FUNCTION_BLOCK FB_Toggle

VAR
	fbTon : TON := (PT := T#10S);
	bStart : BOOL := TRUE;
	fbTof : TOF := (PT := T#10S);
END_VAR

fbTon(IN := bStart);
IF fbTon.Q THEN
	bStart := FALSE;
END_IF
fbTof (IN := bStart);	
IF NOT fbTof.Q	THEN
	bStart := TRUE;
END_IF

END_FUNCTION_BLOCK

(* stored: Version 1.1.0.1, ProductVersion 3.1.4024.16
   POU FB_Toggle: Id {008cb8fd-17f3-4bd0-bd90-3aed1ac4120f}, SpecialFunc None *)
